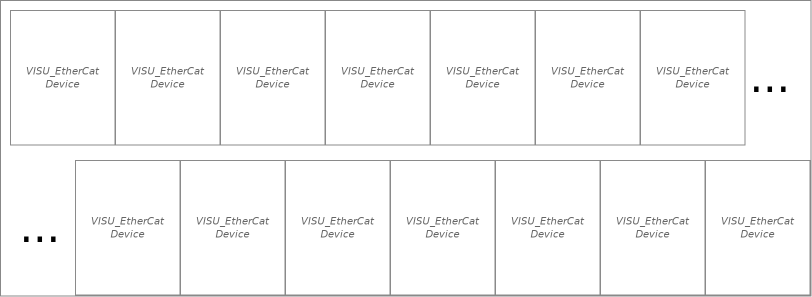
VISUALIZATION VISU_CoverIO  // 812x297
VAR_IN_OUT
	io : CoverIO;
	widget : CoverIOWidget;
END_VAR
    Frame (10,10 105x135)
        shows VISU_EtherCatDevice(device := io.parts.coupler, widget := widget.coupler)
    Label (740,45 60x64), "..."
    Label (10,195 60x64), "..."
    Frame (115,10 105x135)
        shows VISU_EtherCatDevice(device := io.parts.slot1, widget := widget.slot1)
    Frame (220,10 105x135)
        shows VISU_EtherCatDevice(device := io.parts.slot2, widget := widget.slot2)
    Frame (325,10 105x135)
        shows VISU_EtherCatDevice(device := io.parts.slot3, widget := widget.slot3)
    Frame (430,10 105x135)
        shows VISU_EtherCatDevice(device := io.parts.slot4, widget := widget.slot4)
    Frame (535,10 105x135)
        shows VISU_EtherCatDevice(device := io.parts.slot5, widget := widget.slot5)
    Frame (640,10 105x135)
        shows VISU_EtherCatDevice(device := io.parts.slot6, widget := widget.slot6)
    Frame (75,160 105x135)
        shows VISU_EtherCatDevice(device := io.parts.slot7, widget := widget.slot7)
    Frame (180,160 105x135)
        shows VISU_EtherCatDevice(device := io.parts.slot8, widget := widget.slot8)
    Frame (285,160 105x135)
        shows VISU_EtherCatDevice(device := io.parts.slot9, widget := widget.slot9)
    Frame (390,160 105x135)
        shows VISU_EtherCatDevice(device := io.parts.slot10, widget := widget.slot10)
    Frame (495,160 105x135)
        shows VISU_EtherCatDevice(device := io.parts.slot11, widget := widget.slot11)
    Frame (600,160 105x135)
        shows VISU_EtherCatDevice(device := io.parts.slot12, widget := widget.slot12)
    Frame (705,160 105x135)
        shows VISU_EtherCatDevice(device := io.parts.slot13, widget := widget.slot13)
END_VISUALIZATION

(* stored: Version 1.1.0.1, ProductVersion 3.1.4019.2
   Visu VISU_CoverIO: Id {f2a1f0ea-a0ed-4ac9-8917-dc2514413e65} *)
